// TIA Portal project "Filling_Machine" (V14)
// Machine de remplissage

(* hardware
DEVICE "S7-1200 station_1"  S7-1200 Station
   slot 0: "Rack_0"  S7-1200 Rack  Rack  V1.0
   slot 1: "PLC_1"  CPU 1214C DC/DC/DC  6ES7 214-1AG40-0XB0  V4.2
DEVICE "HMI_1"  TP900 Comfort
   slot 0: "TP900 Comfort"  TP900 Comfort  6AV2 124-0JC01-0AX0  14.0.1.0
   slot 1: "HMI_RT_1"  TP900 Comfort  6AV2 124-0JC01-0AX0  14.0.1.0
   slot 5: "HMI_1.IE_CP_1"  PROFINET Interface  14.0.1.0
      slot 1: "PROFINET Interface_1"  PROFINET Interface
         slot 1: "Port_1"  Port
         slot 2: "Port_2"  Port
   slot 7: "HMI_1.MPI/DP_CP_1"  MPI/DP Interface  14.0.1.0
*)

// ===== PLC "PLC_1"  CPU 1214C DC/DC/DC =====

VAR_GLOBAL   // PLC tag table "Default tag table"
   "System_Byte" AT %MB1 : Byte;
   "FirstScan" AT %M1.0 : Bool;
   "DiagStatusUpdate" AT %M1.1 : Bool;
   "AlwaysTRUE" AT %M1.2 : Bool;
   "AlwaysFALSE" AT %M1.3 : Bool;
   "Clock_Byte" AT %MB0 : Byte;
   "Clock_10Hz" AT %M0.0 : Bool;
   "Clock_5Hz" AT %M0.1 : Bool;
   "Clock_2.5Hz" AT %M0.2 : Bool;
   "Clock_2Hz" AT %M0.3 : Bool;
   "Clock_1.25Hz" AT %M0.4 : Bool;
   "Clock_1Hz" AT %M0.5 : Bool;
   "Clock_0.625Hz" AT %M0.6 : Bool;
   "Clock_0.5Hz" AT %M0.7 : Bool;
   "Start_Button" AT %I0.0 : Bool;
   "Stop_Button" AT %I0.1 : Bool;
   "Emergency_Stop" AT %I0.2 : Bool;
   "Proximity_Sensor" AT %I0.3 : Bool;
   "Level_Sensor" AT %I0.4 : Bool;
   "Auto_Manual_Switch" AT %I0.5 : Bool;
   "Tank_Low_Level" AT %I0.6 : Bool;
   "Reset_Button" AT %I0.7 : Bool;
   "Conveyor_Motor" AT %Q0.0 : Bool;
   "Filling_Valve" AT %Q0.1 : Bool;
   "Green_Light" AT %Q0.2 : Bool;
   "Red_Light" AT %Q0.3 : Bool;
   "Orange_Light" AT %Q0.4 : Bool;
   "Buzzer" AT %Q0.5 : Bool;
   "Yellow_Light" AT %Q0.6 : Bool;
   "Pump_Motor" AT %Q0.7 : Bool;
   "Machine_Running" AT %M20.0 : Bool;
   "Filling_Active" AT %M20.1 : Bool;
   "Bottle_Present" AT %M20.2 : Bool;
   "Cycle_Complete" AT %M20.3 : Bool;
   "Auto_Mode" AT %M20.4 : Bool;
   "Manual_Mode" AT %M20.5 : Bool;
   "Conveyor_Start_Delay" AT %M20.6 : Bool;
   "Production_Done" AT %M20.7 : Bool;
   "Alarm_Overflow" AT %M21.0 : Bool;
   "Alarm_No_Bottle" AT %M21.1 : Bool;
   "Alarm_Tank_Empty" AT %M21.2 : Bool;
   "Alarm_Emergency" AT %M21.3 : Bool;
   "HMI_Start" AT %M30.0 : Bool;
   "HMI_Stop" AT %M30.1 : Bool;
   "HMI_Reset" AT %M30.2 : Bool;
   "HMI_Manual_Conveyor" AT %M30.3 : Bool;
   "HMI_Manual_Valve" AT %M30.4 : Bool;
   "HMI_Counter_Reset" AT %M30.5 : Bool;
   "HMI_Manual_Pump" AT %M30.6 : Bool;
   "Edge_Memory_1" AT %M50.0 : Bool;
   "Edge_Memory_2" AT %M50.1 : Bool;
   "Bottle_Counter" AT %MW100 : Int;
   "Production_Target" AT %MW102 : Int;
   "Filling_Time_Set" AT %MW104 : Int;
   "Conveyor_Delay_Set" AT %MW106 : Int;
   "Password_Input" AT %MW200 : Int;
   "Access_Level" AT %MW202 : Int;
   "Login_Success" AT %M40.0 : Bool;
   "HMI_Login_Trigger" AT %M40.2 : Bool;
   "HMI_Logout_Trigger" AT %M40.3 : Bool;
   "Login_Failed" AT %M40.1 : Bool;
   "HMI_Emergency" AT %M30.7 : Bool;
   "HMI_Auto_Mode" AT %M31.0 : Bool;
   "HMI_Bottle_Sensor" AT %M31.1 : Bool;
   "Filling_Timer_Value" AT %MW210 : Int;
   "Filling_Done_Flag" AT %M40.4 : Bool;
   "Cycle_Complete_Reset" AT %M40.5 : Bool;
   "Tag_1" AT %M40.6 : Bool;
END_VAR

// folder: System blocks/Program resources

DATA_BLOCK "IEC_Timer_0_DB"   // DB1
{ S7_Optimized_Access := 'TRUE' }
AUTHOR : Simatic
FAMILY : IEC
NAME : IEC_TMR
VERSION : 1.0
// stored: InstanceOfName IEC_TIMER
"IEC_TIMER"
BEGIN
END_DATA_BLOCK

DATA_BLOCK "IEC_Counter_0_DB"   // DB2
{ S7_Optimized_Access := 'TRUE' }
AUTHOR : Simatic
FAMILY : IEC
NAME : CNTR
VERSION : 1.0
// stored: InstanceOfName IEC_COUNTER
"IEC_COUNTER"
BEGIN
END_DATA_BLOCK

// folder: (top level)

FUNCTION "Login_System" : Void   // FC1, SCL
{ S7_Optimized_Access := 'TRUE' }
VERSION : 0.1
BEGIN
   //===================================================================
   // LOGIN_SYSTEM (FC1) - SCL Function
   // Passwords:
   //   1111 = User (basic access)
   //   9999 = Admin (full access)
   //===================================================================


   // LOGIN BUTTON PRESSED
   IF "HMI_Login_Trigger" THEN

       CASE "Password_Input" OF
           1111:  // USER
               "Access_Level" := 1;
               "Login_Success" := TRUE;
               "Login_Failed" := FALSE;

           9999:  // ADMIN
               "Access_Level" := 2;
               "Login_Success" := TRUE;
               "Login_Failed" := FALSE;

           ELSE:  // WRONG PASSWORD
               "Access_Level" := 0;
               "Login_Success" := FALSE;
               "Login_Failed" := TRUE;
       END_CASE;

       // Reset trigger
       "HMI_Login_Trigger" := FALSE;

   END_IF;


   // LOGOUT BUTTON PRESSED
   IF "HMI_Logout_Trigger" THEN
       "Access_Level" := 0;
       "Login_Success" := FALSE;
       "Login_Failed" := FALSE;
       "Password_Input" := 0;
       "HMI_Logout_Trigger" := FALSE;
   END_IF;


   //===================================================================
   // END OF FC1
   //===================================================================
END_FUNCTION

ORGANIZATION_BLOCK "Main"   // OB1, LAD, ProgramCycle
TITLE = "Main Program Sweep (Cycle)"
{ S7_Optimized_Access := 'TRUE' }
VERSION : 0.1
   VAR_INPUT
      Initial_Call : Bool;   // Initial call of this OB
      Remanence : Bool;   // =True, if remanent data are available
   END_VAR
BEGIN

REGION Network 1: MACHINE START/STOP
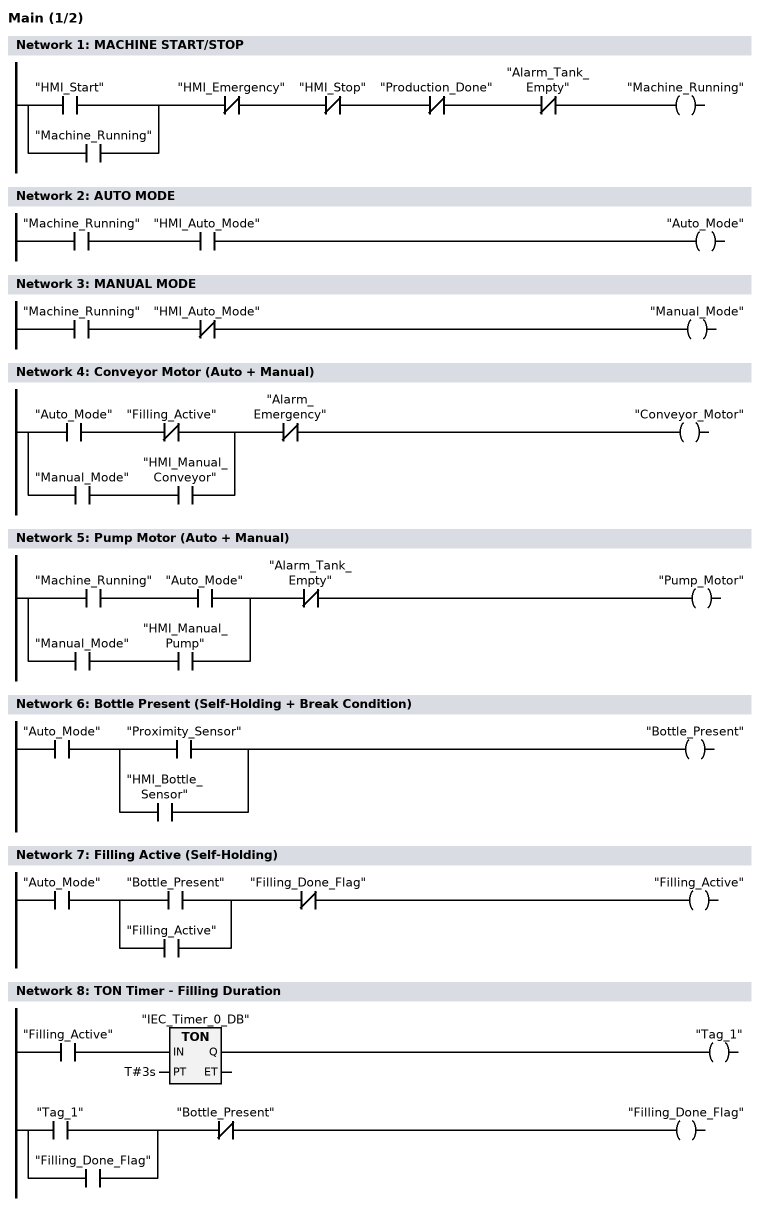
   RUNG wire#powerrail
      Contact( "HMI_Start" )
      wire#w1
      I_Contact( "HMI_Emergency" )
      I_Contact( "HMI_Stop" )
      I_Contact( "Production_Done" )
      I_Contact( "Alarm_Tank_Empty" )
      Coil( "Machine_Running" )
   END_RUNG
   RUNG wire#powerrail
      Contact( "Machine_Running" )
   END_RUNG wire#w1
   // the same network as SCL:
   "Machine_Running" := ("HMI_Start" OR "Machine_Running") AND NOT "HMI_Emergency" AND NOT "HMI_Stop" AND NOT "Production_Done" AND NOT "Alarm_Tank_Empty";
END_REGION

REGION Network 2: AUTO MODE
   RUNG wire#powerrail
      Contact( "Machine_Running" )
      Contact( "HMI_Auto_Mode" )
      Coil( "Auto_Mode" )
   END_RUNG
   // the same network as SCL:
   "Auto_Mode" := "Machine_Running" AND "HMI_Auto_Mode";
END_REGION

REGION Network 3: MANUAL MODE
   RUNG wire#powerrail
      Contact( "Machine_Running" )
      I_Contact( "HMI_Auto_Mode" )
      Coil( "Manual_Mode" )
   END_RUNG
   // the same network as SCL:
   "Manual_Mode" := "Machine_Running" AND NOT "HMI_Auto_Mode";
END_REGION

REGION Network 4: Conveyor Motor (Auto + Manual)
   RUNG wire#powerrail
      Contact( "Auto_Mode" )
      I_Contact( "Filling_Active" )
      wire#w1
      I_Contact( "Alarm_Emergency" )
      Coil( "Conveyor_Motor" )
   END_RUNG
   RUNG wire#powerrail
      Contact( "Manual_Mode" )
      Contact( "HMI_Manual_Conveyor" )
   END_RUNG wire#w1
   // the same network as SCL:
   "Conveyor_Motor" := (("Auto_Mode" AND NOT "Filling_Active") OR ("Manual_Mode" AND "HMI_Manual_Conveyor")) AND NOT "Alarm_Emergency";
END_REGION

REGION Network 5: Pump Motor (Auto + Manual)
   RUNG wire#powerrail
      Contact( "Machine_Running" )
      Contact( "Auto_Mode" )
      wire#w1
      I_Contact( "Alarm_Tank_Empty" )
      Coil( "Pump_Motor" )
   END_RUNG
   RUNG wire#powerrail
      Contact( "Manual_Mode" )
      Contact( "HMI_Manual_Pump" )
   END_RUNG wire#w1
   // the same network as SCL:
   "Pump_Motor" := (("Machine_Running" AND "Auto_Mode") OR ("Manual_Mode" AND "HMI_Manual_Pump")) AND NOT "Alarm_Tank_Empty";
END_REGION

REGION Network 6: Bottle Present (Self-Holding + Break Condition)
   RUNG wire#powerrail
      Contact( "Auto_Mode" )
      wire#w1
      Contact( "Proximity_Sensor" )
      wire#w2
      Coil( "Bottle_Present" )
   END_RUNG
   RUNG wire#w1
      Contact( "HMI_Bottle_Sensor" )
   END_RUNG wire#w2
   // the same network as SCL:
   "Bottle_Present" := "Auto_Mode" AND ("Proximity_Sensor" OR "HMI_Bottle_Sensor");
END_REGION

REGION Network 7: Filling Active (Self-Holding)
   RUNG wire#powerrail
      Contact( "Auto_Mode" )
      wire#w1
      Contact( "Bottle_Present" )
      wire#w2
      I_Contact( "Filling_Done_Flag" )
      Coil( "Filling_Active" )
   END_RUNG
   RUNG wire#w1
      Contact( "Filling_Active" )
   END_RUNG wire#w2
   // the same network as SCL:
   "Filling_Active" := "Auto_Mode" AND ("Bottle_Present" OR "Filling_Active") AND NOT "Filling_Done_Flag";
END_REGION

REGION Network 8: TON Timer - Filling Duration
   "IEC_Timer_0_DB".TON(IN := "Filling_Active", PT := T#3s);
   "Tag_1" := "IEC_Timer_0_DB".Q;
   "Filling_Done_Flag" := ("Tag_1" OR "Filling_Done_Flag") AND NOT "Bottle_Present";
END_REGION

REGION Network 9: Production Done + Counter + Reset
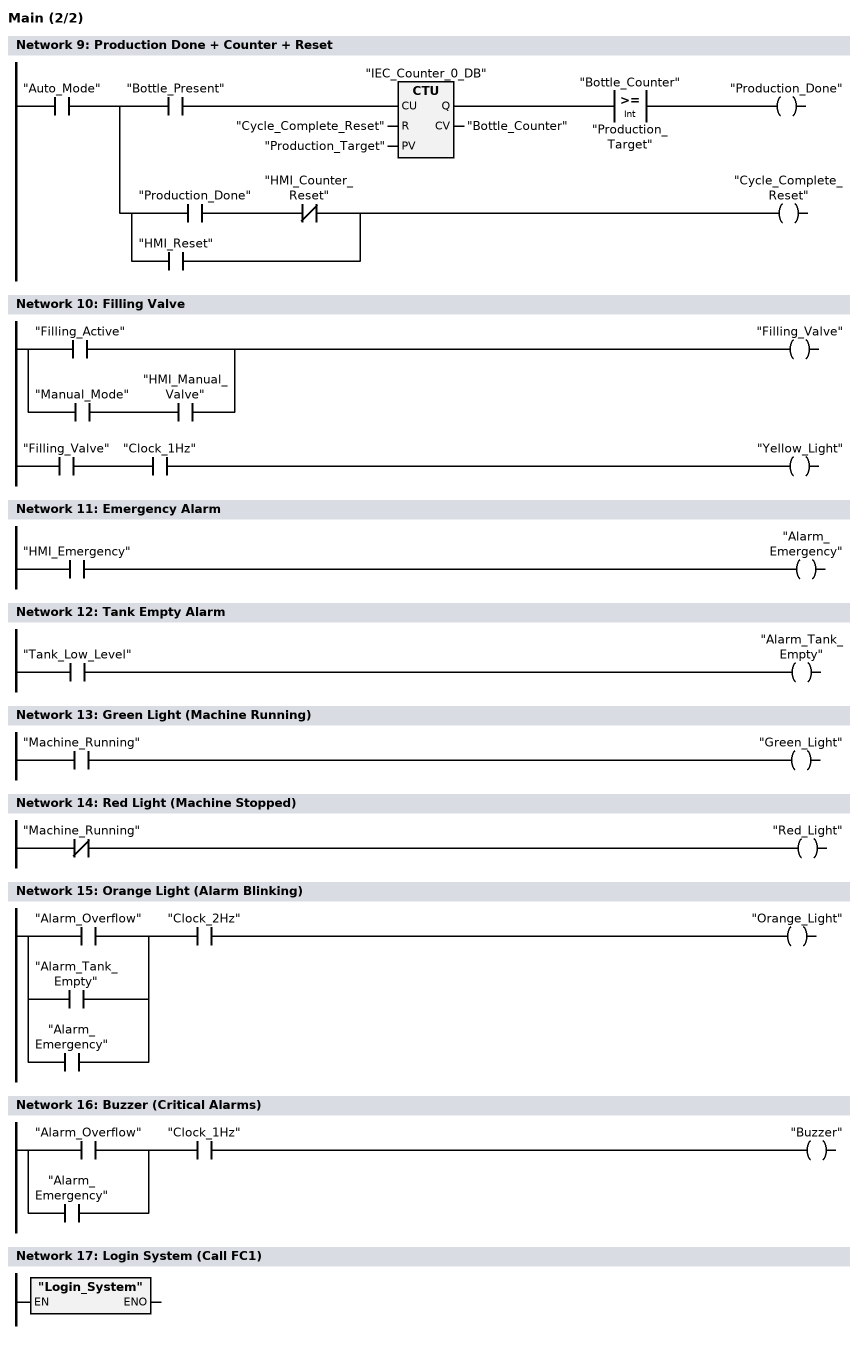
   "IEC_Counter_0_DB".CTU(CU := "Auto_Mode" AND "Bottle_Present",
                          R := "Cycle_Complete_Reset",
                          PV := "Production_Target",
                          CV => "Bottle_Counter");
   "Production_Done" := "IEC_Counter_0_DB".Q AND ("Bottle_Counter" >= "Production_Target");
   "Cycle_Complete_Reset" := "Auto_Mode" AND (("Production_Done" AND NOT "HMI_Counter_Reset") OR "HMI_Reset");
END_REGION

REGION Network 10: Filling Valve
   RUNG wire#powerrail
      Contact( "Filling_Active" )
      wire#w1
      Coil( "Filling_Valve" )
   END_RUNG
   RUNG wire#powerrail
      Contact( "Manual_Mode" )
      Contact( "HMI_Manual_Valve" )
   END_RUNG wire#w1
   RUNG wire#powerrail
      Contact( "Filling_Valve" )
      Contact( "Clock_1Hz" )
      Coil( "Yellow_Light" )
   END_RUNG
   // the same network as SCL:
   "Filling_Valve" := "Filling_Active" OR ("Manual_Mode" AND "HMI_Manual_Valve");
   "Yellow_Light" := "Filling_Valve" AND "Clock_1Hz";
END_REGION

REGION Network 11: Emergency Alarm
   RUNG wire#powerrail
      Contact( "HMI_Emergency" )
      Coil( "Alarm_Emergency" )
   END_RUNG
   // the same network as SCL:
   "Alarm_Emergency" := "HMI_Emergency";
END_REGION

REGION Network 12: Tank Empty Alarm
   RUNG wire#powerrail
      Contact( "Tank_Low_Level" )
      Coil( "Alarm_Tank_Empty" )
   END_RUNG
   // the same network as SCL:
   "Alarm_Tank_Empty" := "Tank_Low_Level";
END_REGION

REGION Network 13: Green Light (Machine Running)
   RUNG wire#powerrail
      Contact( "Machine_Running" )
      Coil( "Green_Light" )
   END_RUNG
   // the same network as SCL:
   "Green_Light" := "Machine_Running";
END_REGION

REGION Network 14: Red Light (Machine Stopped)
   RUNG wire#powerrail
      I_Contact( "Machine_Running" )
      Coil( "Red_Light" )
   END_RUNG
   // the same network as SCL:
   "Red_Light" := NOT "Machine_Running";
END_REGION

REGION Network 15: Orange Light (Alarm Blinking)
   RUNG wire#powerrail
      Contact( "Alarm_Overflow" )
      wire#w1
      Contact( "Clock_2Hz" )
      Coil( "Orange_Light" )
   END_RUNG
   RUNG wire#powerrail
      Contact( "Alarm_Tank_Empty" )
   END_RUNG wire#w1
   RUNG wire#powerrail
      Contact( "Alarm_Emergency" )
   END_RUNG wire#w1
   // the same network as SCL:
   "Orange_Light" := ("Alarm_Overflow" OR "Alarm_Tank_Empty" OR "Alarm_Emergency") AND "Clock_2Hz";
END_REGION

REGION Network 16: Buzzer (Critical Alarms)
   RUNG wire#powerrail
      Contact( "Alarm_Overflow" )
      wire#w1
      Contact( "Clock_1Hz" )
      Coil( "Buzzer" )
   END_RUNG
   RUNG wire#powerrail
      Contact( "Alarm_Emergency" )
   END_RUNG wire#w1
   // the same network as SCL:
   "Buzzer" := ("Alarm_Overflow" OR "Alarm_Emergency") AND "Clock_1Hz";
END_REGION

REGION Network 17: Login System (Call FC1)
   RUNG wire#powerrail
      "Login_System"()
   END_RUNG
   // the same network as SCL:
   "Login_System"();
END_REGION
END_ORGANIZATION_BLOCK

(* ===== HMI "HMI_RT_1" =====
system functions are stored by id; their names below are inferred from use
connection "HMI_Connection_1": ETHERNET, S7_1200_OMS

HMI tags "Default tag table"
   "System_Byte" : Byte = PLC System_Byte AT %MB1, 1 s
   "FirstScan" : Bool = PLC FirstScan AT %M1.0, 1 s
   "DiagStatusUpdate" : Bool = PLC DiagStatusUpdate AT %M1.1, 1 s
   "AlwaysTRUE" : Bool = PLC AlwaysTRUE AT %M1.2, 1 s
   "AlwaysFALSE" : Bool = PLC AlwaysFALSE AT %M1.3, 1 s
   "Clock_Byte" : Byte = PLC Clock_Byte AT %MB0, 1 s
   "Clock_10Hz" : Bool = PLC Clock_10Hz AT %M0.0, 1 s
   "Clock_5Hz" : Bool = PLC Clock_5Hz AT %M0.1, 1 s
   "Clock_2.5Hz" : Bool = PLC "Clock_2.5Hz" AT %M0.2, 1 s
   "Clock_2Hz" : Bool = PLC Clock_2Hz AT %M0.3, 1 s
   "Clock_1.25Hz" : Bool = PLC "Clock_1.25Hz" AT %M0.4, 1 s
   "Clock_1Hz" : Bool = PLC Clock_1Hz AT %M0.5, 1 s
   "Clock_0.625Hz" : Bool = PLC "Clock_0.625Hz" AT %M0.6, 1 s
   "Clock_0.5Hz" : Bool = PLC "Clock_0.5Hz" AT %M0.7, 1 s
   "Start_Button" : Bool = PLC Start_Button AT %I0.0, 1 s
   "Stop_Button" : Bool = PLC Stop_Button AT %I0.1, 1 s
   "Emergency_Stop" : Bool = PLC Emergency_Stop AT %I0.2, 1 s
   "Proximity_Sensor" : Bool = PLC Proximity_Sensor AT %I0.3, 1 s
   "Level_Sensor" : Bool = PLC Level_Sensor AT %I0.4, 1 s
   "Auto_Manual_Switch" : Bool = PLC Auto_Manual_Switch AT %I0.5, 1 s
   "Tank_Low_Level" : Bool = PLC Tank_Low_Level AT %I0.6, 1 s
   "Reset_Button" : Bool = PLC Reset_Button AT %I0.7, 1 s
   "Conveyor_Motor" : Bool = PLC Conveyor_Motor AT %Q0.0, 1 s
   "Filling_Valve" : Bool = PLC Filling_Valve AT %Q0.1, 1 s
   "Green_Light" : Bool = PLC Green_Light AT %Q0.2, 1 s
   "Red_Light" : Bool = PLC Red_Light AT %Q0.3, 1 s
   "Orange_Light" : Bool = PLC Orange_Light AT %Q0.4, 1 s
   "Buzzer" : Bool = PLC Buzzer AT %Q0.5, 1 s
   "Yellow_Light" : Bool = PLC Yellow_Light AT %Q0.6, 1 s
   "Pump_Motor" : Bool = PLC Pump_Motor AT %Q0.7, 1 s
   "Machine_Running" : Bool = PLC Machine_Running AT %M20.0, 1 s
   "Filling_Active" : Bool = PLC Filling_Active AT %M20.1, 1 s
   "Bottle_Present" : Bool = PLC Bottle_Present AT %M20.2, 1 s
   "Cycle_Complete" : Bool = PLC Cycle_Complete AT %M20.3, 1 s
   "Auto_Mode" : Bool = PLC Auto_Mode AT %M20.4, 1 s
   "Manual_Mode" : Bool = PLC Manual_Mode AT %M20.5, 1 s
   "Conveyor_Start_Delay" : Bool = PLC Conveyor_Start_Delay AT %M20.6, 1 s
   "Production_Done" : Bool = PLC Production_Done AT %M20.7, 1 s
   "Alarm_Overflow" : Bool = PLC Alarm_Overflow AT %M21.0, 1 s
   "Alarm_No_Bottle" : Bool = PLC Alarm_No_Bottle AT %M21.1, 1 s
   "Alarm_Tank_Empty" : Bool = PLC Alarm_Tank_Empty AT %M21.2, 1 s
   "Alarm_Emergency" : Bool = PLC Alarm_Emergency AT %M21.3, 1 s
   "HMI_Start" : Bool = PLC HMI_Start AT %M30.0, 1 s
   "HMI_Stop" : Bool = PLC HMI_Stop AT %M30.1, 1 s
   "HMI_Reset" : Bool = PLC HMI_Reset AT %M30.2, 1 s
   "HMI_Manual_Conveyor" : Bool = PLC HMI_Manual_Conveyor AT %M30.3, 1 s
   "HMI_Manual_Valve" : Bool = PLC HMI_Manual_Valve AT %M30.4, 1 s
   "HMI_Counter_Reset" : Bool = PLC HMI_Counter_Reset AT %M30.5, 1 s
   "HMI_Manual_Pump" : Bool = PLC HMI_Manual_Pump AT %M30.6, 1 s
   "Edge_Memory_1" : Bool = PLC Edge_Memory_1 AT %M50.0, 1 s
   "Edge_Memory_2" : Bool = PLC Edge_Memory_2 AT %M50.1, 1 s
   "Bottle_Counter" : Int = PLC Bottle_Counter AT %MW100, 1 s
   "Production_Target" : Int = PLC Production_Target AT %MW102, 1 s
   "Filling_Time_Set" : Int = PLC Filling_Time_Set AT %MW104, 1 s
   "Password_Input" : Int = PLC Password_Input AT %MW200, 1 s
   "Access_Level" : Int = PLC Access_Level AT %MW202, 1 s
   "Login_Success" : Bool = PLC Login_Success AT %M40.0, 1 s
   "Login_Failed" : Bool = PLC Login_Failed AT %M40.1, 1 s
   "HMI_Login_Trigger" : Bool = PLC HMI_Login_Trigger AT %M40.2, 1 s
   "HMI_Logout_Trigger" : Bool = PLC HMI_Logout_Trigger AT %M40.3, 1 s
   "HMI_Emergency" : Bool = PLC HMI_Emergency AT %M30.7, 1 s
   "HMI_Auto_Mode" : Bool = PLC HMI_Auto_Mode AT %M31.0, 1 s
   "HMI_Bottle_Sensor" : Bool = PLC HMI_Bottle_Sensor AT %M31.1, 1 s
   "Filling_Timer_Value" : Int = PLC Filling_Timer_Value AT %MW210, 1 s

text list "Status_Text_List": 0 'STOPPED'; 1 'RUNNING'

text list "Mode_Text_List": 0 'MANUAL'; 1 'AUTO'

text list "Alarm_Status_List": 0 '[ Inactive ]'; 1 '[ ACTIVE ]'

text list "Access_Level_List": 0 'NOT LOGGED IN'; 1 'USER'; 2 'ADMIN'

text list "Login_Status_List": 0 '-- Waiting --'; 1 'SUCCESS'

screen "Root screen" 800x480
   TextField "Text field_1" at 10,5 size 500x40; Text 'FILLING MACHINE - MAIN SCREEN'
   Button "Button_1" at 680,8 size 100x35; TextOff '☰ MENU'
      on Click: ActivateScreen("Menu_Screen", 0)
   TextField "Text field_2" at 30,78 size 230x25; Text 'MACHINE STATUS'
   Circle "Circle_1" at 58,115 size 20x20
      Appearance <- "Machine_Running"
   TextField "Text field_3" at 88,115 size 80x20; Text 'Machine:'
   SymbolicIOField "Symbolic I/O field_1" at 178,113 size 100x25; TextOff '0'; TextOn '1'; TextList "Status_Text_List"
      ProcessValue <- "Machine_Running"
   Circle "Circle_2" at 58,152 size 20x20
      Appearance <- "Auto_Mode"
   TextField "Text field_4" at 88,152 size 80x20; Text 'Mode:'
   SymbolicIOField "Symbolic I/O field_2" at 178,150 size 100x25; TextOn '1'; TextOff '0'; TextList "Mode_Text_List"
      ProcessValue <- "Auto_Mode"
   TextField "Text field_5" at 490,78 size 230x25; Text 'COUNTERS'
   TextField "Text field_6" at 516,108 size 110x25; Text 'Bottles Filled:'
   IOField "I/O field_1" at 624,105 size 109x30; FormatPattern 9999
      ProcessValue <- "Bottle_Counter"
   TextField "Text field_7" at 520,147 size 110x25; Text 'Target:'
   IOField "I/O field_2" at 624,143 size 110x30; FormatPattern 9999
      ProcessValue <- "Production_Target"
      ObjectEnable <- "Access_Level"
   TextField "Text field_8" at 30,206 size 230x25; Text 'MACHINE VIEW'
   GraphicView "Graphic view_10" at 104,260 size 128x141; Picture "Graphic_11"
   GraphicView "Graphic view_1" at 158,249 size 20x17; Picture "Graphic_13"
   GraphicView "Graphic view_3" at 177,228 size 88x20; Picture "Graphic_16"
   GraphicView "Graphic view_2" at 157,226 size 23x26; Picture "Graphic_14"
   GraphicView "Graphic view_5" at 315,216 size 195x20; Picture "Graphic_16"
   GraphicView "Graphic view_7" at 508,234 size 20x17; Picture "Graphic_13"
   GraphicView "Graphic view_8" at 325,350 size 389x48; Picture "Graphic_23"
   GraphicView "Graphic view_4" at 262,217 size 57x41; Picture "Graphic_17"
   GraphicView "Graphic view_9" at 508,215 size 21x23; Picture "Graphic_31"
   GraphicView "Graphic view_11" at 507,284 size 20x32; Picture "Graphic_33"
   GraphicView "Graphic view_6" at 504,249 size 33x39; Picture "Graphic_19"
   GraphicView "Graphic view_12" at 503,319 size 28x55; Picture "Graphic_29"
   GraphicView "Graphic view_13" at 138,291 size 61x61; Picture "Graphic_34"
   Circle "Circle_3" at 283,263 size 16x16
      Appearance <- "Pump_Motor"
   Circle "Circle_4" at 542,262 size 16x16
      Appearance <- "Filling_Valve"
   TextField "Text field_9" at 299,261 size 50x20; Text 'Pump'
   TextField "Text field_10" at 558,261 size 50x20; Text 'Valve'
   TextField "Text field_11" at 113,239 size 50x20; Text 'Tank'
   Rectangle "Rectangle_7" at 507,337 size 21x33
      Visibility <- "Filling_Active"
   GraphicView "Graphic view_15" at 336,379 size 16x16; Picture "Graphic_36"
      Visibility <- "Conveyor_Motor"
   GraphicView "Graphic view_14" at 336,379 size 16x16; Picture "Graphic_35"
      Visibility <- "Conveyor_Motor"
   GraphicView "Graphic view_16" at 351,379 size 16x16; Picture "Graphic_36"
      Visibility <- "Conveyor_Motor"
   GraphicView "Graphic view_17" at 351,379 size 16x16; Picture "Graphic_35"
      Visibility <- "Conveyor_Motor"
   GraphicView "Graphic view_18" at 366,379 size 16x16; Picture "Graphic_36"
      Visibility <- "Conveyor_Motor"
   GraphicView "Graphic view_19" at 366,379 size 16x16; Picture "Graphic_35"
      Visibility <- "Conveyor_Motor"
   GraphicView "Graphic view_20" at 381,379 size 16x16; Picture "Graphic_36"
      Visibility <- "Conveyor_Motor"
   GraphicView "Graphic view_21" at 381,379 size 16x16; Picture "Graphic_35"
      Visibility <- "Conveyor_Motor"
   GraphicView "Graphic view_22" at 396,379 size 16x16; Picture "Graphic_36"
      Visibility <- "Conveyor_Motor"
   GraphicView "Graphic view_23" at 396,379 size 16x16; Picture "Graphic_35"
      Visibility <- "Conveyor_Motor"
   GraphicView "Graphic view_24" at 411,379 size 16x16; Picture "Graphic_36"
      Visibility <- "Conveyor_Motor"
   GraphicView "Graphic view_25" at 411,379 size 16x16; Picture "Graphic_35"
      Visibility <- "Conveyor_Motor"
   GraphicView "Graphic view_26" at 427,379 size 16x16; Picture "Graphic_36"
      Visibility <- "Conveyor_Motor"
   GraphicView "Graphic view_27" at 427,379 size 16x16; Picture "Graphic_35"
      Visibility <- "Conveyor_Motor"
   GraphicView "Graphic view_28" at 443,379 size 16x16; Picture "Graphic_36"
      Visibility <- "Conveyor_Motor"
   GraphicView "Graphic view_29" at 443,379 size 16x16; Picture "Graphic_35"
      Visibility <- "Conveyor_Motor"
   GraphicView "Graphic view_30" at 459,379 size 16x16; Picture "Graphic_36"
      Visibility <- "Conveyor_Motor"
   GraphicView "Graphic view_31" at 459,379 size 16x16; Picture "Graphic_35"
      Visibility <- "Conveyor_Motor"
   GraphicView "Graphic view_32" at 475,379 size 16x16; Picture "Graphic_36"
      Visibility <- "Conveyor_Motor"
   GraphicView "Graphic view_33" at 475,379 size 16x16; Picture "Graphic_35"
      Visibility <- "Conveyor_Motor"
   GraphicView "Graphic view_34" at 491,379 size 16x16; Picture "Graphic_36"
      Visibility <- "Conveyor_Motor"
   GraphicView "Graphic view_35" at 491,379 size 16x16; Picture "Graphic_35"
      Visibility <- "Conveyor_Motor"
   GraphicView "Graphic view_36" at 505,379 size 16x16; Picture "Graphic_36"
      Visibility <- "Conveyor_Motor"
   GraphicView "Graphic view_37" at 505,379 size 16x16; Picture "Graphic_35"
      Visibility <- "Conveyor_Motor"
   GraphicView "Graphic view_38" at 521,379 size 16x16; Picture "Graphic_36"
      Visibility <- "Conveyor_Motor"
   GraphicView "Graphic view_39" at 521,379 size 16x16; Picture "Graphic_35"
      Visibility <- "Conveyor_Motor"
   GraphicView "Graphic view_40" at 535,379 size 16x16; Picture "Graphic_36"
      Visibility <- "Conveyor_Motor"
   GraphicView "Graphic view_41" at 535,379 size 16x16; Picture "Graphic_35"
      Visibility <- "Conveyor_Motor"
   GraphicView "Graphic view_42" at 549,379 size 16x16; Picture "Graphic_36"
      Visibility <- "Conveyor_Motor"
   GraphicView "Graphic view_43" at 549,379 size 16x16; Picture "Graphic_35"
      Visibility <- "Conveyor_Motor"
   GraphicView "Graphic view_44" at 565,379 size 16x16; Picture "Graphic_36"
      Visibility <- "Conveyor_Motor"
   GraphicView "Graphic view_45" at 565,379 size 16x16; Picture "Graphic_35"
      Visibility <- "Conveyor_Motor"
   GraphicView "Graphic view_46" at 581,379 size 16x16; Picture "Graphic_36"
      Visibility <- "Conveyor_Motor"
   GraphicView "Graphic view_47" at 581,379 size 16x16; Picture "Graphic_35"
      Visibility <- "Conveyor_Motor"
   GraphicView "Graphic view_48" at 597,379 size 16x16; Picture "Graphic_36"
      Visibility <- "Conveyor_Motor"
   GraphicView "Graphic view_49" at 597,379 size 16x16; Picture "Graphic_35"
      Visibility <- "Conveyor_Motor"
   GraphicView "Graphic view_50" at 613,379 size 16x16; Picture "Graphic_36"
      Visibility <- "Conveyor_Motor"
   GraphicView "Graphic view_51" at 613,379 size 16x16; Picture "Graphic_35"
      Visibility <- "Conveyor_Motor"
   GraphicView "Graphic view_52" at 628,379 size 16x16; Picture "Graphic_36"
      Visibility <- "Conveyor_Motor"
   GraphicView "Graphic view_53" at 628,379 size 16x16; Picture "Graphic_35"
      Visibility <- "Conveyor_Motor"
   Button "Button_2" at 50,431 size 160x32; TextOff 'START'
      on Press: SetBit("HMI_Start")
      on Release: InvertBit("HMI_Start")
      ObjectEnable <- "Access_Level"
   Button "Button_3" at 230,431 size 160x32; TextOff 'STOP'
      ObjectEnable <- "Access_Level"
      on Click: InvertBit("HMI_Stop")
      on Press: InvertBit("HMI_Stop")
   Button "Button_4" at 410,431 size 160x32; TextOff 'RESET'
      ObjectEnable <- "Access_Level"
      on Press: SetBit("HMI_Reset")
      on Release: InvertBit("HMI_Reset")
   Button "Button_5" at 590,431 size 160x32; TextOff 'RESET COUNTER'
      ObjectEnable <- "Access_Level"
      on Press: SetBit("HMI_Counter_Reset")
      on Release: InvertBit("HMI_Counter_Reset")
   Button "Button_6" at 350,71 size 100x49; TextOff 'EMERGENCY'
      on Click: InvertBit("HMI_Emergency")
      Appearance <- "HMI_Emergency"
   Button "Button_7" at 350,129 size 100x55; TextOff 'MODE MANUAL'
      on Click: InvertBit("HMI_Auto_Mode")
      Visibility <- "HMI_Auto_Mode"
   Button "Button_8" at 645,214 size 100x70; TextOff 'BOTTLE'
      Appearance <- "HMI_Bottle_Sensor"
      on Press: SetBit("HMI_Bottle_Sensor")
      on Release: InvertBit("HMI_Bottle_Sensor")
   Button "Button_9" at 350,129 size 100x55; TextOff 'MODE MANUAL'
      on Click: InvertBit("HMI_Auto_Mode")
      Visibility <- "HMI_Auto_Mode"

screen "Menu_Screen" 800x480
   TextField "Text field_1" at 250,10 size 300x30; Text 'NAVIGATION MENU'
   Button "Button_1" at 70,100 size 200x140; TextOff 'MAIN'
      on Click: ActivateScreen("Root screen", 0)
   Button "Button_2" at 300,100 size 200x140; TextOff 'MANUAL'
      on Click: ActivateScreen("Manual_Screen", 0)
   Button "Button_3" at 530,100 size 200x140; TextOff 'SETTINGS'
      on Click: ActivateScreen("Settings_Screen", 0)
   Button "Button_4" at 70,270 size 200x140; TextOff 'ALARMS'
      on Click: ActivateScreen("Alarms_Screen", 0)
   Button "Button_5" at 300,270 size 200x140; TextOff 'TRENDS'
      on Click: ActivateScreen("Trends_Screen", 0)
   Button "Button_6" at 530,270 size 200x140; TextOff 'LOGOUT'
      on Click: ActivateScreen("Login_Screen", 0)

screen "Manual_Screen" 800x480
   TextField "Text field_1" at 10,5 size 500x40; Text 'MANUAL CONTROL'
   Button "Button_1" at 680,10 size 100x35; TextOff '☰ MENU'
      on Click: ActivateScreen("Menu_Screen", 0)
   TextField "Text field_2" at 285,80 size 230x25; Text 'CURRENT MODE:'
   SymbolicIOField "Symbolic I/O field_1" at 285,110 size 230x30; TextOff '0'; TextOn '1'; TextList "Mode_Text_List"
      ProcessValue <- "Auto_Mode"
   TextField "Text field_3" at 30,180 size 400x25; Text 'MANUAL EQUIPMENT CONTROL'
   TextField "Text field_4" at 60,230 size 200x25; Text 'CONVEYOR'
   Button "Button_2" at 90,270 size 140x50; TextOff 'ON / OFF'
      on Press: SetBit("HMI_Manual_Conveyor")
      on Release: ResetBit("HMI_Manual_Conveyor")
      ObjectEnable <- "Access_Level"
   TextField "Text field_6" at 60,340 size 70x25; Text 'Status:'
   SymbolicIOField "Symbolic I/O field_2" at 140,340 size 90x25; TextOff '0'; TextOn '1'; TextList "Status_Text_List"
      ProcessValue <- "Conveyor_Motor"
   TextField "Text field_5" at 300,230 size 200x25; Text 'VALVE'
   Button "Button_3" at 330,270 size 140x50; TextOff 'ON / OFF'
      on Release: ResetBit("HMI_Manual_Valve")
      on Press: SetBit("HMI_Manual_Valve")
      ObjectEnable <- "Access_Level"
   TextField "Text field_7" at 300,340 size 70x25; Text 'Status:'
   SymbolicIOField "Symbolic I/O field_3" at 380,340 size 90x25; TextOn '1'; TextOff '0'; TextList "Status_Text_List"
      ProcessValue <- "Filling_Valve"
   TextField "Text field_8" at 540,230 size 200x25; Text 'PUMP'
   Button "Button_4" at 570,270 size 140x50; TextOff 'ON / OFF'
      on Release: ResetBit("HMI_Manual_Pump")
      on Press: SetBit("HMI_Manual_Pump")
      ObjectEnable <- "Access_Level"
   TextField "Text field_9" at 540,340 size 70x25; Text 'Status:'
   SymbolicIOField "Symbolic I/O field_4" at 620,340 size 90x25; TextOn '1'; TextOff '0'; TextList "Status_Text_List"
      ProcessValue <- "Pump_Motor"
   TextField "Text field_10" at 20,430 size 760x30; Text 'Warning: Manual controls work ONLY when Auto/Manual switch is in MANUAL position'

screen "Settings_Screen" 800x480
   TextField "Text field_1" at 10,5 size 500x40; Text 'SETTINGS'
   Button "Button_1" at 680,10 size 100x35; TextOff '☰ MENU'
      on Click: ActivateScreen("Menu_Screen", 0)
   TextField "Text field_2" at 30,80 size 300x25; Text 'PRODUCTION SETTINGS'
   TextField "Text field_3" at 50,120 size 200x30; Text 'Production Target:'
   IOField "I/O field_1" at 280,118 size 120x35; FormatPattern 9999
      ProcessValue <- "Production_Target"
      ObjectEnable <- "Access_Level"
   TextField "Text field_4" at 420,120 size 80x30; Text 'bottles'
   TextField "Text field_5" at 50,165 size 200x30; Text 'Max Filling Time:'
   IOField "I/O field_2" at 280,163 size 120x35; FormatPattern 9999
      ProcessValue <- "Filling_Time_Set"
      ObjectEnable <- "Access_Level"
   TextField "Text field_6" at 420,163 size 80x30; Text 'seconds'
   TextField "Text field_7" at 30,290 size 300x25; Text 'COUNTER MANAGEMENT'
   TextField "Text field_8" at 50,330 size 180x30; Text 'Current Counter:'
   IOField "I/O field_3" at 250,328 size 120x35; FormatPattern 9999
      ProcessValue <- "Bottle_Counter"
   TextField "Text field_9" at 390,330 size 80x30; Text 'bottles'
   Button "Button_2" at 520,325 size 220x45; TextOff 'RESET COUNTER'
      on Press: SetBit("HMI_Reset")
      on Release: InvertBit("HMI_Reset")
      ObjectEnable <- "Access_Level"
   TextField "Text field_10" at 20,440 size 760x25; Text 'Note: Changes are saved automatically when you press Enter'

screen "Alarms_Screen" 800x480
   TextField "Text field_1" at 10,5 size 500x40; Text 'ALARMS'
   Button "Button_1" at 680,10 size 100x35; TextOff '☰ MENU'
      on Click: ActivateScreen("Menu_Screen", 0)
   TextField "Text field_2" at 30,80 size 300x25; Text 'ACTIVE ALARMS'
   Ellipse "Ellipse_1" at 50,120 size 20x20
      Appearance <- "Alarm_Emergency"
   TextField "Text field_3" at 110,121 size 37x20; Text 'Text'
   TextField "Text field_4" at 90,120 size 300x25; Text 'EMERGENCY STOP'
   SymbolicIOField "Symbolic I/O field_1" at 265,120 size 130x32; TextOff '0'; TextOn '1'; TextList "Alarm_Status_List"
      ProcessValue <- "Alarm_Emergency"
   Ellipse "Ellipse_2" at 50,155 size 20x20
      Appearance <- "Alarm_Tank_Empty"
   TextField "Text field_5" at 90,155 size 300x25; Text 'TANK EMPTY'
   SymbolicIOField "Symbolic I/O field_2" at 265,155 size 130x32; TextOn '1'; TextOff '0'; TextList "Alarm_Status_List"
      ProcessValue <- "Alarm_Tank_Empty"
   Ellipse "Ellipse_3" at 50,190 size 20x20
      Appearance <- "Alarm_Overflow"
   TextField "Text field_6" at 90,190 size 300x25; Text 'OVERFLOW'
   SymbolicIOField "Symbolic I/O field_3" at 265,190 size 130x32; TextOn '1'; TextOff '0'; TextList "Alarm_Status_List"
      ProcessValue <- "Alarm_Overflow"
   Ellipse "Ellipse_4" at 50,225 size 20x20
      Appearance <- "Alarm_No_Bottle"
   TextField "Text field_7" at 90,225 size 300x25; Text 'NO BOTTLE'
   SymbolicIOField "Symbolic I/O field_4" at 265,225 size 130x32; TextOn '1'; TextOff '0'; TextList "Alarm_Status_List"
      ProcessValue <- "Alarm_No_Bottle"
   TextField "Text field_8" at 30,310 size 300x25; Text 'ALARM SUMMARY'
   TextField "Text field_9" at 30,345 size 720x25; Text 'Emergency Stop is a critical alarm - Machine cannot start until released'
   Button "Button_2" at 280,410 size 240x50; TextOff 'RESET ALARMS'
      on Press: SetBit("HMI_Reset")
      on Release: InvertBit("HMI_Reset")
      ObjectEnable <- "Access_Level"

screen "Trends_Screen" 800x480
   TextField "Text field_1" at 10,5 size 500x40; Text 'TRENDS'
   Button "Button_1" at 680,10 size 100x35; TextOff '☰ MENU'
      on Click: ActivateScreen("Menu_Screen", 0)
   TrendView "Trend view_1" at 20,70 size 760x290
   TextField "Text field_2" at 30,388 size 200x25; Text 'STATISTICS'
   TextField "Text field_3" at 50,420 size 70x25; Text 'Total:'
   IOField "I/O field_1" at 130,418 size 80x28; FormatPattern 9999
      ProcessValue <- "Bottle_Counter"
   TextField "Text field_4" at 240,420 size 70x25; Text 'Target:'
   TextField "Text field_5" at 440,420 size 70x25; Text 'Access:'
   IOField "I/O field_2" at 320,418 size 80x28; FormatPattern 9999
      ProcessValue <- "Production_Target"
   SymbolicIOField "Symbolic I/O field_1" at 520,418 size 200x28; TextOff '0'; TextOn '1'
      ProcessValue <- "Access_Level"

screen "Login_Screen" 800x480
   TextField "Text field_1" at 10,5 size 500x40; Text 'LOGIN'
   Button "Button_1" at 680,10 size 100x35; TextOff '☰ MENU'
      on Click: ActivateScreen("Menu_Screen", 0)
   TextField "Text field_2" at 210,115 size 380x35; Text 'USER LOGIN'
   TextField "Text field_3" at 230,170 size 150x25; Text 'Access Level:'
   Button "Button_2" at 230,259 size 160x60; TextOff 'LOGIN'
      on Click: SetBit("HMI_Login_Trigger")
   Button "Button_3" at 410,259 size 160x60; TextOff 'LOGOUT'
      on Press: SetBit("HMI_Logout_Trigger")
      on Release: InvertBit("HMI_Logout_Trigger")
   SymbolicIOField "Symbolic I/O field_1" at 390,170 size 180x30; TextOff '0'; TextOn '1'; TextList "Access_Level_List"
      ProcessValue <- "Access_Level"
   TextField "Text field_4" at 230,210 size 150x25; Text 'Password:'
   IOField "I/O field_1" at 390,208 size 180x30; FormatPattern 9999
      ProcessValue <- "Password_Input"
   TextField "Text field_6" at 230,340 size 100x25; Text 'Status:'
   SymbolicIOField "Symbolic I/O field_2" at 340,340 size 200x30; TextOff '0'; TextOn '1'; TextList "Login_Status_List"
      ProcessValue <- "Login_Success"
   TextField "Text field_5" at 230,390 size 340x60; Text 'Passwords: • 1111 = User (Basic) • 9999 = Admin (Full)'
*)